Universal Robots PolyScope program: trigger_reduced_mode_208.urp

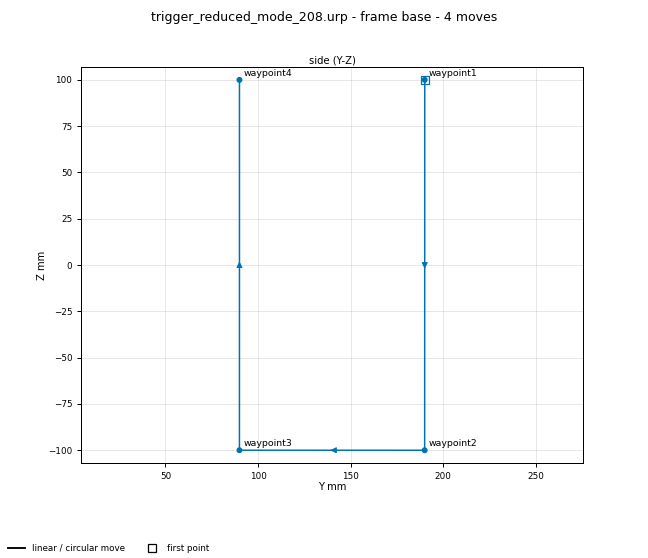
[picture p0: tool path of trigger_reduced_mode_208.urp in frame base, 4 of 4 moves have a stored position in this frame; points joined in program order, loops and branches not executed]
Program trigger_reduced_mode_208 (createdIn=3.2.19293 lastSavedIn=3.2.19293 directory=/programs installation=default robotSerialNumber=2015351391)
Calibrated DH parameters: a=[0.000352, -0.161198, -0.373486, 0.00005, 0.000049, 0]; d=[0.089268, 352.477598, -320.08558, -32.281492, 0.094939, 0.082518]; alpha=[1.570728, 0.001116, -0.003686, 1.571189, -1.570572, 0]; deltaTheta=[-0.000012, 1.181849, -1.491165, 0.309495, -0.000007, 0.000025]
Robot Program (runOnlyOnce=false motionType=MoveJ speed=1.047198 acceleration=1.396263 recalculateMotions=false)
  MoveL speed 1500 mm/s, acceleration 2500 mm/s^2 (recalculateMotions=false) feature=Base
    Waypoint waypoint1: TCP in base x=372.372 y=190.044 z=100.015 mm, rx=-0.0046 ry=-3.1392 rz=0.1204 rad; joints [44.083, -87.256, -123.682, -62.149, 86.65, 134.188] deg; flange x=372.403 y=199.62 z=224.632 mm, rx=-0.0046 ry=-3.1391 rz=0.1204 rad
    Waypoint waypoint2: TCP in base x=372.346 y=189.995 z=-100.045 mm, rx=-0.0045 ry=-3.1391 rz=0.1208 rad; joints [44.096, -114.097, -134.59, -24.394, 86.792, 134.113] deg; flange x=372.389 y=199.64 z=24.633 mm, rx=-0.0046 ry=-3.1391 rz=0.1204 rad
    Waypoint waypoint3: TCP in base x=372.348 y=89.953 z=-100.035 mm, rx=-0.0046 ry=-3.1391 rz=0.1207 rad; joints [32.565, -111.65, -140.64, -20.1, 86.25, 122.577] deg; flange x=372.39 y=99.583 z=24.619 mm, rx=-0.0046 ry=-3.1392 rz=0.1205 rad
    Waypoint waypoint4: TCP in base x=372.381 y=89.97 z=99.993 mm, rx=-0.0046 ry=-3.1392 rz=0.1206 rad; joints [32.55, -81.604, -128.836, -61.953, 86.097, 122.651] deg; flange x=372.395 y=99.569 z=224.632 mm, rx=-0.0046 ry=-3.1392 rz=0.1205 rad
